// RPC calls are not allowed in Local mode.
IF stat.bLocal THEN
	RPC_MoveRel	:= M_SetRpcStatus(E_SA_RPC_ERROR.LOCAL);
	RETURN;
// Move Relative command is accepted only in OP state.
ELSIF	stat.nState <> E_SA_POS_ELT_STATE.OP	THEN
	RPC_MoveRel	:= M_SetRpcStatus(E_SA_RPC_ERROR.NOT_OP);
	RETURN;
// The positioner has to be initialised / OP (operational), i.e. already REFerenced.
ELSIF	NOT stat.bInitialised	THEN
	RPC_MoveRel	:= M_SetRpcStatus(E_SA_RPC_ERROR.CH_NOT_OP);
	RETURN;
// Set velocity cannot be 0.0.
ELSIF	in_lrVel = 0.0	THEN
	RPC_MoveRel	:= M_SetRpcStatus(E_SA_RPC_ERROR.VEL_ZERO);
	RETURN;
// Set velocity cannot be < 0.0.
ELSIF	in_lrVel <= 0.0	THEN
	RPC_MoveRel	:= M_SetRpcStatus(E_SA_RPC_ERROR.VEL_NEG);
	RETURN;
// Set velocity cannot be greater than MAX Velocity.
ELSIF	in_lrVel > cfg.lrMaxVelocity	THEN
	RPC_MoveRel	:= M_SetRpcStatus(E_SA_RPC_ERROR.VEL_MAX);
	RETURN;
// If SW limits are active, check the limits
ELSIF cfg.lrRangeLimitMax > cfg.lrRangeLimitMin THEN
	IF lrPos < cfg.lrRangeLimitMin THEN
		RPC_MoveRel	:= M_SetRpcStatus(E_SA_RPC_ERROR.SW_LIMIT_LOWER);
		RETURN;
	ELSIF lrPos > cfg.lrRangeLimitMax THEN
		RPC_MoveRel	:= M_SetRpcStatus(E_SA_RPC_ERROR.SW_LIMIT_UPPER);
		RETURN;
	END_IF
END_IF

// Set command
ctrl.nCmd	:= E_SA_CH_CMD.MOV;
ctrl.lrPos	:= lrPos;
ctrl.lrVel	:= in_lrVel;


// Call was successful
RPC_MoveRel	:= M_SetRpcStatus(E_SA_RPC_ERROR.OK);
END_METHOD

{attribute 'TcRpcEnable':='1'}
METHOD RPC_Reset : INT
VAR_INPUT
END_VAR
// If the SmarAct MCS2 Controller is in error,
// the positioner cannot be controlled.
IF stat.nCtrlErrorCode <> 0  OR  stat.nCtrlState <> E_RS_BASE_STATE.OP THEN
	RPC_Reset	:= M_SetRpcStatus(E_SA_RPC_ERROR.CTRL_ERROR);
	RETURN;
END_IF


// RPC calls are not allowed in Local mode.
IF stat.bLocal THEN
	RPC_Reset	:= M_SetRpcStatus(E_SA_RPC_ERROR.LOCAL);
	RETURN;
END_IF

// Cannot RESET positioner while moving.
IF stat.nState = E_SA_POS_ELT_STATE.OP  AND  stat.nSubstate = E_SA_POS_ELT_SUBSTATE.OP_MOVING  THEN
	RPC_Reset	:= M_SetRpcStatus(E_SA_RPC_ERROR.MOVING);
	RETURN;
END_IF


// Set command
ctrl.nCmd	:= E_SA_CH_CMD.RESET;

//stat.nState			:= E_SA_POS_ELT_STATE.NONE;
//stat.nSubstate		:= E_SA_POS_ELT_SUBSTATE.NONE;


// Call was successful
RPC_Reset	:= M_SetRpcStatus(E_SA_RPC_ERROR.OK);
END_METHOD

{attribute 'TcRpcEnable':='1'}
METHOD RPC_Stop : INT
VAR_INPUT
END_VAR
// If the SmarAct MCS2 Controller is in error,
// the positioner cannot be controlled.
IF stat.nCtrlErrorCode <> 0  OR  stat.nCtrlState <> E_RS_BASE_STATE.OP THEN
	RPC_Stop	:= M_SetRpcStatus(E_SA_RPC_ERROR.CTRL_ERROR);
	RETURN;
END_IF


// RPC calls are not allowed in Local mode.
IF stat.bLocal THEN
	RPC_Stop	:= M_SetRpcStatus(E_SA_RPC_ERROR.LOCAL);
	RETURN;
END_IF


// Set STOP command
ctrl.nCmd	:= E_SA_CH_CMD.STOP;

// Call was successful
RPC_Stop	:= M_SetRpcStatus(E_SA_RPC_ERROR.OK);
END_METHOD

END_FUNCTION_BLOCK

// ---- POUs/F_GetRpcErrorText.TcPOU
FUNCTION F_GetRpcErrorText : STRING
VAR_INPUT
	ErrorCode:	INT;
END_VAR
VAR
	str:	STRING;
END_VAR

CASE ErrorCode OF
	E_SA_RPC_ERROR.OK:					str	:= 'OK';
	E_SA_RPC_ERROR.NOT_OP:				str	:= 'Positioner not OPERATIONAL';
	E_SA_RPC_ERROR.NOT_NOTOP_READY:		str	:= 'Call failed. Not in NOTOP_READY.';
	E_SA_RPC_ERROR.NOT_NOTOP_NOTREADY:	str	:= 'Call failed. Not in NOTOP_NOTREADY/ERROR.';
	E_SA_RPC_ERROR.LOCAL:				str	:= 'RPC calls not allowed in Local mode.';
	E_SA_RPC_ERROR.SW_LIMIT_LOWER:		str	:= 'Target position beyond Lower SW Limit';
	E_SA_RPC_ERROR.SW_LIMIT_UPPER:		str	:= 'Target position beyond Upper SW Limit';
	E_SA_RPC_ERROR.CHANNEL:				str	:= 'Channel not in range [0..17]';
	E_SA_RPC_ERROR.VEL_MAX:				str	:= 'Target Velocity higher than Maximum';
	E_SA_RPC_ERROR.VEL_NEG:				str	:= 'Target Velocity cannot be negative';
	E_SA_RPC_ERROR.VEL_ZERO:			str	:= 'Target Velocity cannot be zero';
	E_SA_RPC_ERROR.CH_NOT_OP:			str	:= 'Channel not OPERATIONAL. REFerence first.';
	E_SA_RPC_ERROR.CTRL_ERROR:			str	:= 'SmarAct MCS2 Controller Problem';
	E_SA_RPC_ERROR.MOVING:				str	:= 'Positioner is moving. Stop first.';
	E_SA_RPC_ERROR.COMM:				str	:= 'SmarAct MCS2 Controller Communication Problem';
ELSE
	str	:= 'Unregistered RPC error.';
END_CASE

F_GetRpcErrorText	:= str;

END_FUNCTION

// ---- POUs/F_STRING_TO_LINT.TcPOU
FUNCTION F_STRING_TO_LINT : LINT
VAR_INPUT
	in_s:	STRING;
END_VAR
VAR
	lrVal:	LREAL;
END_VAR

// STRING_TO_LINT DOES NOT WORK !!!!!
//
// The string has to be converted to LREAL first and then to LINT
//
lrVal	:= STRING_TO_LREAL(in_s);

F_STRING_TO_LINT	:= LREAL_TO_LINT(lrVal);

END_FUNCTION

// ---- Examples/FB_SA_CH_PDS_IRIS.TcPOU
FUNCTION_BLOCK FB_SA_CH_PDS_IRIS EXTENDS FB_SA_CHANNEL_BASE
VAR_INPUT
END_VAR
VAR_OUTPUT
END_VAR
VAR
END_VAR

//
// SID-50 specific non-linear conversion 
// from Device units [nd] to user units [%] of opening.
//
METHOD M_ConvertPosDev2User : LREAL
VAR_INPUT
	lnDevValue:	LINT;
END_VAR
VAR
	lrDiam:	LREAL;		// Diameter of opening [mm].
END_VAR
//
// Note that iris increases the opening when moving in negative direction.
// That's why the scale is negative in the configuration.
// Linear conversion implemented in M_ConvertDev2User().
// UU   = DevU / scale * BASE_RES
// DevU = UU   * scale / BASE_RES
//
lrDiam	:= M_ConvertDev2User(lnDevValue);

//
// Maximum opening is 50 mm.
// Current opening is relative to that.
//    % = diam^2 / 50^2 * 100.0
//
M_ConvertPosDev2User := (lrDiam * lrDiam) / (50.0 * 50.0) * 100.0;
END_METHOD

//
// SID-50 specific non-linear conversion 
// from user units [%] of opening to Device units [nd].
//
METHOD M_ConvertPosUser2Dev : LINT
VAR_INPUT
	lrUserValue:	LREAL;	// Percentage of opening
END_VAR
VAR
	lrDiam:	LREAL;		// Diameter of opening [mm].
END_VAR
//
// Note that iris increases the opening when moveng in negative direction.
// That's why the scale is negative in the configuration.
//

//
// Get the opening diameter from the percentage relative to 50 mm for SID-50.
//    % = lrUserValue;
//    % = 100.0 * diam^2 / 50^2  ==> diam = SQRT(% / 100.0 * 50^2)
//
lrDiam	:= SQRT(lrUserValue / 100.0 * 50.0 * 50.0);

//
// Convert diameter to device unitd - linear conversion.
//
M_ConvertPosUser2Dev := M_ConvertUser2Dev(lrDiam);
END_METHOD

END_FUNCTION_BLOCK

// ---- Examples/FB_SMARACT_SIM.TcPOU
FUNCTION_BLOCK FB_SMARACT_SIM EXTENDS FB_SMAR_ACT_BASE
VAR_INPUT
END_VAR
VAR_OUTPUT
END_VAR
VAR
	//
	// TODO USER: Add existing SmarAct Positioners
	//
	// We use prefix 'x_' just for the convenience that
	// all positioners appear together in the OPC UA Namespace.
	//
	x_fw1:	FB_SA_CHANNEL_BASE;	// CH 0
	x_fw2:	FB_SA_CHANNEL_BASE;	// CH 1
	x_iris:	FB_SA_CH_PDS_IRIS;	// CH 2 non-linear scaling for % of opening
END_VAR

//
// Execute the base class object FB_SMAR_ACT_BASE.
//
SUPER^();

METHOD M_ConfigureUser
VAR_INPUT
END_VAR
VAR
	i:		UINT;
	nMod:	UINT;	// Module number
	
END_VAR
//
// This method defines specific configurations for each positioner/channel.
//

// 
// In this example, three positioners are defined in FB_SMARACT_SIM.
//
//	fw1:	FB_SA_CHANNEL_BASE;
//	fw2:	FB_SA_CHANNEL_BASE;
//	iris:	FB_SA_CHANNEL_BASE;
//

//
// Configure used channels [0..17].
// In this example, there are three used channels: 0, 1 and 2.
//
cfg.arrUsedCh[0]	:= TRUE;
cfg.arrUsedCh[1]	:= TRUE;
cfg.arrUsedCh[2]	:= TRUE;


//
// Set pointers to instances of used channels
//
ptrCH[0]	:= ADR(x_fw1);
ptrCH[1]	:= ADR(x_fw2);
ptrCH[2]	:= ADR(x_iris);


//
// Initial configuration of each exiting positioner.
//

//
// SFW-6-25.4 - Filter Wheel 1
//
x_fw1.M_Configure(
	in_sName			:= 'Filter Wheel - 1',
	in_sUnits			:= 'deg',
	in_lrScale			:= 1.0, 
	in_lrREF_POS		:= 60.0,	// REF mark pos
	in_lrREF_VEL		:= 20.0,	// Velocity for referencing [UU/s]
	in_nHOLD			:= -1,		// Hold infinitely
	in_lrINP_THR		:= 0.001,	// in-pos threshold = 0.001 deg
	in_nINP_DEL			:= 500,		// in-pos delay 500 ms
	in_lrMaxVelocity	:= 30,		// Maximum permitted Velocity
	in_lrRangeLimitMin	:= 0.0,		// Min=Max ==> No limits
	in_lrRangeLimitMax	:= 0.0,		// Min=Max ==> No limits 
	in_nREF_OPT			:= 0,		// Referencing in positive direction
	in_nCAL_OPT			:= 0,		// Calibrating in positive direction
	in_nPCON_OPT		:= 256);	// 'in-pos' flag set

//
// SFW-6-25.4 - Filter Wheel 2
//
x_fw2.M_Configure(
	in_sName			:= 'Filter Wheel - 2',
	in_sUnits			:= 'deg',
	in_lrScale			:= 1.0, 
	in_lrREF_POS		:= 120.0,	// REF mark pos
	in_lrREF_VEL		:= 20.0,	// Velocity for referencing [UU/s]
	in_nHOLD			:= -1,		// Hold infinitely
	in_lrINP_THR		:= 0.001,	// in-pos threshold = 0.001 deg
	in_nINP_DEL			:= 1000,	// in-pos delay 500 ms
	in_lrMaxVelocity	:= 30,		// Maximum permitted Velocity
	in_lrRangeLimitMin	:= 0.0,		// Min=Max ==> No limits
	in_lrRangeLimitMax	:= 0.0,		// Min=Max ==> No limits 
	in_nREF_OPT			:= 0,		// Referencing in positive direction
	in_nCAL_OPT			:= 0,		// Calibrating in positive direction
	in_nPCON_OPT		:= 256);	// 'in-pos' flag set

//
// SID-50 - Iris Diaphragm
//
// Note: Because the scale is negative, MIN and MAX values are swapped.
//       In Device Units, the diaphragm will move between -5..-50 (/scale) mm.
//       In User   Units, the diaphragm will move between 1..100 %.
//
// The position of the diaphragm is the percentage of the opening.
//

x_iris.M_Configure(
	in_sName			:= 'SHAPS Diaphragm',
	in_sUnits			:= '%',
	in_lrScale			:= -0.001763245, 
	in_lrREF_POS		:= 34.33,	// REF mark pos in %. (Diam = 29.29832067 mm)
	in_lrREF_VEL		:= 5.0,		// Velocity for referencing [UU/s]
	in_nHOLD			:= -1,		// Hold infinitely
	in_lrINP_THR		:= 0.0005,	// in-pos threshold = 0.0005 %
	in_nINP_DEL			:= 500,		// in-pos delay 500 ms
	in_lrMaxVelocity	:= 15,		// Maximum permitted Velocity
	in_lrRangeLimitMin	:= 100.001,	// Min limit (positive because in_lrScale < 0) !!!
	in_lrRangeLimitMax	:= 0.999,	// Max limit (negative because in_lrScale < 0) !!!
	in_nREF_OPT			:= 0,		// Referencing in positive direction
	in_nCAL_OPT			:= 0,		// Calibrating in positive direction
	in_nPCON_OPT		:= 256);	// 'in-pos' flag set
END_METHOD

END_FUNCTION_BLOCK

// ---- POUs/Simulation/FB_SIM_SMAR_ACT.TcPOU
FUNCTION_BLOCK FB_SIM_SMAR_ACT EXTENDS FB_SIM_TCP_DEVICE_BASE
VAR_INPUT
END_VAR
VAR_OUTPUT
END_VAR
VAR
	arrCH:		ARRAY [0..17] OF FB_SIM_SA_CHANNEL;
	i:			UINT;
END_VAR

IF NOT in_bEnable THEN
	RETURN;
ELSE
	//
	// Execute instance of the simulator
	//
	Device(	in_bSimulation	:= in_bSimulation,
			in_sTcpIpAdr	:= in_sTcpIpAdr,
			in_nTcpPort		:= in_nTcpPort);
	
	//
	// Execute State Machine for each instance Channel simulator.
	//
	FOR i:=0 TO 17 DO
		arrCH[i].M_StateMachine();
	END_FOR
			
	//
	// Check for received commands.
	//
	IF Device.out_bAccepted AND Device.out_bReceived THEN
		// A command has arrived. Send a simulated reply
		sReply	:=	M_GetSimReply(in_sReceived	:=Device.out_sReceived); 
		
		// Trigger SEND only if there is a reply
		IF sReply <> ''	THEN
			ptrDevCtrl^.nCommand	:= E_RS_COMM_CMD.SEND;
			ptrDevCtrl^.sCmd		:= sReply;
			ptrDevCtrl^.bExecute	:= TRUE;
		END_IF
	END_IF
END_IF

METHOD M_GetSimReply : STRING(255)
VAR_INPUT
	{attribute 'OPC.UA.DA' := '0'}
	in_sReceived:	STRING(255);		// String received from a client
END_VAR
VAR
	sReply:	STRING(255);
	sTmp:	STRING;
	sTmp2:	STRING;
	lrVal:	LREAL;
	nValue:	UINT;
	i:		INT;
    fbFormat   : FB_FormatString;
    sOut       : T_MaxString;
	nCh:	UINT;	// Channel number
	nPos:	INT;	// Position in the string

	lnVel:	LINT;	// MOVE Velocity
	lnPos:	LINT;	// MOVE Target Position
END_VAR
//
// Commands related to the controller/DEVice
//
IF FIND (in_sReceived, '*IDN?') > 0 THEN
	// MCS2 ID
	M_GetSimReply	:= CONCAT('SIM SmarAct;MCS2-00005855;MCS2-00005855;07/05/21', in_sReplySuffix);

ELSIF FIND (in_sReceived, ':DEV:SNUM?') > 0 THEN
	// MCS2 S/N
	M_GetSimReply	:= CONCAT('"MCS2-00005855"', in_sReplySuffix);

ELSIF FIND (in_sReceived, ':DEV:STAT?') > 0 THEN
	// MCS2 State
	// 16 => Only stDevState.bGLOBAL_INPUT set to TRUE.
	M_GetSimReply	:= CONCAT('16', in_sReplySuffix);

//
// Replies to commands starting with ':MOD'.
//
ELSIF FIND(in_sReceived, ':MOD') = 1 THEN
	IF FIND(in_sReceived, ':STAT?') > 1 THEN
		// MOD state is 1 - BIT_SM_PRESENT.
		M_GetSimReply	:= CONCAT('1', in_sReplySuffix);
	END_IF

ELSE
	//
	// Commands related to individual channels
	//
	IF	FIND (in_sReceived, ':CHAN') = 1	THEN
			// Get the channel number that comes 
			// after ':CHAN', e.g. ':CHAN2:STAT?'
			sTmp	:= DELETE(in_sReceived,5,1);
			nCh		:= STRING_TO_UINT(sTmp);
			// The string looks like '2:STAT?' now.
			// Remove the channel number and the following ':' from the command,
			// i.e. remove '2:' and pass 'STAT?' to the channel.
			nPos	:= FIND (sTmp, ':');
			sTmp	:= DELETE(sTmp,nPos,1);
			sReply	:= arrCH[nCH].M_GetChSimReply(sTmp);
			IF sReply <> ''	THEN
				// There is a reply from the channel.
				// Channel reply doesn't contain the reply suffix. Add it.
				M_GetSimReply	:= CONCAT(sReply, in_sReplySuffix);
			ELSE
				// Channel Reply is empty string.
				// Don't reply, i.e. reply is empty string.
				M_GetSimReply	:= '';
			END_IF
	ELSIF	FIND (in_sReceived, ':REF') = 1	THEN
			// Get the channel number that comes 
			// after ':REF' , e.g. ':REF2'
			sTmp	:= DELETE(in_sReceived,4,1);
			nCh		:= STRING_TO_UINT(sTmp);
			arrCH[nCH].M_StartREF();
			M_GetSimReply	:= '';	// No reply to this command
	ELSIF	FIND (in_sReceived, ':CAL') = 1		THEN
			// Get the channel number that comes 
			// after ':CAL', e.g. ':CAL2'
			sTmp	:= DELETE(in_sReceived,4,1);
			nCh		:= STRING_TO_UINT(sTmp);
			arrCH[nCH].M_StartCAL();
			M_GetSimReply	:= '';	// No reply to this command
	ELSIF	FIND (in_sReceived, ':MOVE') = 1	THEN
			// Get the channel number that comes 
			// after ':MOVE', in e.g. ':MOVE2 100000'
			sTmp	:= DELETE(in_sReceived,5,1);	// '2 100000'
			nCh		:= STRING_TO_UINT(sTmp);
			// Find the space and delete everything up to and including the space.
			nPos	:= FIND (sTmp, ' ');
			sTmp2	:= DELETE(sTmp, nPos, 1);	// '100000'
			lnPos	:= F_STRING_TO_LINT(sTmp2);	// Target Position
			lnVel	:= arrCH[nCH].ctrl.lnVEL;	// Target Velocity
			arrCH[nCH].M_StartMOVE(lnPos, lnVel);
			M_GetSimReply	:= '';	// No reply to this command
	ELSIF	FIND (in_sReceived, ':STOP') = 1	THEN
			// Get the channel number that comes 
			// after ':MOVE', e.g. ':MOVE2'
			sTmp	:= DELETE(in_sReceived,5,1);
			nCh		:= STRING_TO_UINT(sTmp);
			arrCH[nCH].M_STOP();
			M_GetSimReply	:= '';	// No reply to this command
	END_IF
END_IF
END_METHOD

END_FUNCTION_BLOCK

// ---- POUs/Simulation/FB_SIM_SA_CHANNEL.TcPOU
FUNCTION_BLOCK FB_SIM_SA_CHANNEL
VAR_INPUT
END_VAR
VAR_OUTPUT
END_VAR
VAR
	cfg:	T_SA_SIM_CH_CFG;
	ctrl:	T_SA_SIM_CH_CTRL;
	stat:	T_SA_SIM_CH_STATUS;
	
	fbTimer:		TON;

END_VAR

// Execute State Machine
M_StateMachine();

METHOD M_GetChSimReply : STRING(255)
VAR_INPUT
	{attribute 'OPC.UA.DA' := '0'}
	in_sCmd:	STRING(255);		// String received from a client
END_VAR
VAR
	sReply:	STRING(255);
	sTmp:	STRING;
	lrVal:	LREAL;
	nValue:	UINT;
	i:		INT;
    fbFormat   : FB_FormatString;
    sOut       : T_MaxString;
	nCh:	INT := 8;	// Number of channels for models 218 and 224
END_VAR

IF FIND (in_sCmd, '?') > 0 THEN
	// This is a query command.
	// There is a reply.
	// Check commands one by one.

	IF FIND (in_sCmd, 'STAT?') > 0 THEN
		// Channel state
		M_GetChSimReply	:= UDINT_TO_STRING(stat.nSTATE);
	ELSIF FIND (in_sCmd, 'CAL:OPT?') > 0 THEN
		// Channel state
		M_GetChSimReply	:= UINT_TO_STRING(cfg.nCAL_OPT);
	ELSIF FIND (in_sCmd, 'REF:OPT?') > 0 THEN
		// Channel state
		M_GetChSimReply	:= UINT_TO_STRING(cfg.nREF_OPT);
	ELSIF FIND (in_sCmd, 'PCON:OPT?') > 0 THEN
		// Channel Positioner control otions
		M_GetChSimReply	:= UINT_TO_STRING(cfg.nPCON_OPT);
	ELSIF FIND (in_sCmd, 'INP:THR?') > 0 THEN
		// Channel in-position threshold
		M_GetChSimReply	:= UDINT_TO_STRING(cfg.nINP_THR);
	ELSIF FIND (in_sCmd, 'INP:DEL?') > 0 THEN
		// Channel in-position delay
		M_GetChSimReply	:= UDINT_TO_STRING(cfg.nINP_DEL);
	ELSIF FIND (in_sCmd, 'RLIM:MIN?') > 0 THEN
		// Channel Limit Min
		M_GetChSimReply	:= LINT_TO_STRING(cfg.lnRLIM_MIN);
	ELSIF FIND (in_sCmd, 'RLIM:MAX?') > 0 THEN
		// Channel Limit Max
		M_GetChSimReply	:= LINT_TO_STRING(cfg.lnRLIM_MAX);
	ELSIF FIND (in_sCmd, 'POS:TARG?') > 0 THEN
		// Channel target position
		M_GetChSimReply	:= LINT_TO_STRING(stat.lnPosTarget);
	ELSIF FIND (in_sCmd, 'POS:CURR?') > 0 THEN
		// Channel actual position
		M_GetChSimReply	:= LINT_TO_STRING(stat.lnPosActual);
	ELSIF FIND (in_sCmd, 'CLIN?') > 0 THEN
		// Channel 
		M_GetChSimReply	:= DINT_TO_STRING(cfg.nCLIN);
	ELSIF FIND (in_sCmd, 'TUN:BASE:UNIT?') > 0 THEN
		// Channel 
		M_GetChSimReply	:= DINT_TO_STRING(cfg.nBASE_UNIT);
	ELSIF FIND (in_sCmd, 'TUN:BASE:RES?') > 0 THEN
		// Channel 
		M_GetChSimReply	:= DINT_TO_STRING(cfg.nBASE_RES);
	ELSIF FIND (in_sCmd, 'TUN:MTYP?') > 0 THEN
		// Channel 
		M_GetChSimReply	:= DINT_TO_STRING(cfg.nTUN_MTYP);
	ELSIF FIND (in_sCmd, 'TUN:RTYP?') > 0 THEN
		// Channel 
		M_GetChSimReply	:= LINT_TO_STRING(cfg.nTUN_RTYP);
	END_IF
ELSE
	// This is a control command.
	// There is NO reply.
	// BUT there are some action to be taken

	IF FIND (in_sCmd, 'CAL:OPT ') > 0 THEN
		// Get the value
		sTmp			:= DELETE(in_sCmd,8,1);
		cfg.nCAL_OPT	:= STRING_TO_UINT(sTmp);
	ELSIF FIND (in_sCmd, 'REF:OPT ') > 0 THEN
		// Get the value
		sTmp			:= DELETE(in_sCmd,8,1);
		cfg.nREF_OPT	:= STRING_TO_UINT(sTmp);
	ELSIF FIND (in_sCmd, 'PCON:OPT ') > 0 THEN
		// Get the value
		sTmp			:= DELETE(in_sCmd,9,1);
		cfg.nPCON_OPT	:= STRING_TO_UINT(sTmp);
	ELSIF FIND (in_sCmd, 'INP:THR ') > 0 THEN
		// Get the value
		sTmp			:= DELETE(in_sCmd,8,1);
		cfg.nINP_THR	:= STRING_TO_UDINT(sTmp);
	ELSIF FIND (in_sCmd, 'INP:DEL ') > 0 THEN
		// Get the value
		sTmp			:= DELETE(in_sCmd,8,1);
		cfg.nINP_DEL	:= STRING_TO_UDINT(sTmp);
	ELSIF FIND (in_sCmd, 'RLIM:MIN ') > 0 THEN
		// Get the value
		sTmp			:= DELETE(in_sCmd,9,1);
		cfg.lnRLIM_MIN	:= STRING_TO_UINT(sTmp);
	ELSIF FIND (in_sCmd, 'RLIM:MAX ') > 0 THEN
		// Get the value
		sTmp			:= DELETE(in_sCmd,9,1);
		cfg.lnRLIM_MAX	:= STRING_TO_UINT(sTmp);
	ELSIF FIND (in_sCmd, 'POS:TARG ') > 0 THEN
		// Get the value
		sTmp			:= DELETE(in_sCmd,9,1);
		stat.lnPosTarget:= F_STRING_TO_LINT(sTmp);
	ELSIF FIND (in_sCmd, 'POS:CURR ') > 0 THEN
		// Get the value
		sTmp			:= DELETE(in_sCmd,9,1);
		stat.lnPosActual:= F_STRING_TO_LINT(sTmp);
	ELSIF FIND (in_sCmd, 'VEL ') > 0 THEN
		// Get the value
		sTmp			:= DELETE(in_sCmd,4,1);
		cfg.lnVEL		:= F_STRING_TO_LINT(sTmp);
		ctrl.lnVEL		:= F_STRING_TO_LINT(sTmp);
	ELSIF FIND (in_sCmd, 'POS ') > 0 THEN
		// Get the value
		sTmp			:= DELETE(in_sCmd,4,1);
		stat.lnPosActual:= F_STRING_TO_LINT(sTmp);
	END_IF
	
	// There is no reply to control commands !!!
	M_GetChSimReply	:= '';
END_IF
END_METHOD

METHOD M_StartCAL
VAR_INPUT
END_VAR
// Start CALibration simulation
;
END_METHOD

METHOD M_StartMOVE
VAR_INPUT
	in_lnPos:	LINT;	// Target Position
	in_lnVel:	LINT;	// Target Velocity
END_VAR
VAR 
	nState:		UDINT := 0;
	nTime:		UDINT :=0;	// Calculated move time [ms].
END_VAR
// Start MOVE simulation

// Set target velocity and position.
ctrl.lnVEL			:= in_lnVel;
ctrl.lnPOS			:= in_lnPos;
stat.lnPosTarget	:= in_lnPos;
stat.lnPosStart		:= stat.lnPosActual;	// MOVE started from this position

// Get the distance to move.
// If distance is zero, do nothing.
stat.lnDistance	:= ctrl.lnPOS - stat.lnPosActual;
IF stat.lnDistance = 0	THEN
	// No movement
	fbTimer(IN:=FALSE);
	RETURN;
END_IF

nState	:= nState OR E_SA_CH_STATE.BIT_ACTIVELY_MOVING;
nState	:= nState OR E_SA_CH_STATE.BIT_CLOSED_LOOP_ACTIVE;
nState	:= nState OR E_SA_CH_STATE.BIT_SENSOR_PRESENT;
nState	:= nState OR E_SA_CH_STATE.BIT_IS_CALIBRATED;
nState	:= nState OR E_SA_CH_STATE.BIT_IS_REFERENCED;
nState	:= nState OR E_SA_CH_STATE.BIT_AMPLIFIER_ENABLED;

stat.nSTATE	:= nState;

// Get time [ms] needed for the move
IF in_lnVel = 0	THEN
	nTime	:= 1000;
ELSE	
	nTime	:= LINT_TO_UDINT(1000 * ABS(stat.lnDistance) / in_lnVel);
END_IF

IF nTime > 0 THEN
	// Set the positioner State Machine State
	stat.nPosState	:=	E_SA_POS_SM_STATE.MOVING;
	
	// Start the timer.
	// Simulated REFerencing should finish in 5 sec.
	fbTimer(IN:=FALSE);
	fbTimer(IN:=TRUE,PT:=UDINT_TO_TIME(nTime));
ELSE
	// No movement
	fbTimer(IN:=FALSE);
END_IF
END_METHOD

METHOD M_StartREF
VAR_INPUT
END_VAR
VAR 
	nState:		UDINT := 0;
END_VAR
// Start REFerencing simulation

nState	:= nState OR E_SA_CH_STATE.BIT_ACTIVELY_MOVING;
nState	:= nState OR E_SA_CH_STATE.BIT_CLOSED_LOOP_ACTIVE;
nState	:= nState OR E_SA_CH_STATE.BIT_REFERENCING;
nState	:= nState OR E_SA_CH_STATE.BIT_SENSOR_PRESENT;
nState	:= nState OR E_SA_CH_STATE.BIT_AMPLIFIER_ENABLED;

stat.nSTATE	:= nState;

// Set the positioner State Machine State
stat.nPosState	:=	E_SA_POS_SM_STATE.CALIB_REF;

// Start the timer.
// Simulated REFerencing should finish in 5 sec.
fbTimer(IN:=FALSE);
fbTimer(IN:=TRUE,PT:=T#5S);
END_METHOD

METHOD M_StateMachine
VAR_INPUT
END_VAR
VAR 
	nState:		UDINT := 0;
	lrProgress:	LREAL;		// Movement progress [0.0..1.0]
	lnPosInc:	LINT;		// Position increment from starting position.
END_VAR
// Execute the timer.
fbTimer();

CASE stat.nPosState OF
	E_SA_POS_SM_STATE.CALIB_REF:
		// Check if referencing is complete.
		IF fbTimer.Q THEN
			// Reset timer
			fbTimer(IN:=FALSE);
			// Set flags for completed REFerencing
			nState	:= nState OR E_SA_CH_STATE.BIT_CLOSED_LOOP_ACTIVE;
			nState	:= nState OR E_SA_CH_STATE.BIT_SENSOR_PRESENT;
			nState	:= nState OR E_SA_CH_STATE.BIT_IS_CALIBRATED;
			nState	:= nState OR E_SA_CH_STATE.BIT_IS_REFERENCED;
			nState	:= nState OR E_SA_CH_STATE.BIT_REFERENCE_MARK;
			nState	:= nState OR E_SA_CH_STATE.BIT_AMPLIFIER_ENABLED;
			nState	:= nState OR E_SA_CH_STATE.BIT_IN_POSITION;
			
			stat.nSTATE	:= nState;
			
			// Set the calibrated position
			stat.lnPosTarget	:= cfg.lnREF_POS;
			stat.lnPosActual	:= cfg.lnREF_POS;
			
			// Set the positioner State Machine State
			stat.nPosState	:=	E_SA_POS_SM_STATE.OP;
		END_IF
	E_SA_POS_SM_STATE.MOVING:
		// Simulate movement progress
		IF fbTimer.PT = T#0MS THEN
			RETURN;
		END_IF
		lrProgress	:= TIME_TO_LREAL(fbTimer.ET) / TIME_TO_LREAL(fbTimer.PT);
		lnPosInc	:= LREAL_TO_LINT(LINT_TO_LREAL(stat.lnDistance) * lrProgress);
		stat.lnPosActual	:= stat.lnPosStart + lnPosInc;
		
		// Check if the move is complete.
		IF fbTimer.Q THEN
			// Reset timer
			fbTimer(IN:=FALSE);
			// Set flags for completed REFerencing
			nState	:= nState OR E_SA_CH_STATE.BIT_CLOSED_LOOP_ACTIVE;
			nState	:= nState OR E_SA_CH_STATE.BIT_SENSOR_PRESENT;
			nState	:= nState OR E_SA_CH_STATE.BIT_IS_CALIBRATED;
			nState	:= nState OR E_SA_CH_STATE.BIT_IS_REFERENCED;
			nState	:= nState OR E_SA_CH_STATE.BIT_AMPLIFIER_ENABLED;
			nState	:= nState OR E_SA_CH_STATE.BIT_IN_POSITION;
			
			stat.nSTATE	:= nState;
			
			// Set the positioner State Machine State
			stat.nPosState	:=	E_SA_POS_SM_STATE.OP;
		END_IF
END_CASE
END_METHOD

METHOD M_STOP
VAR_INPUT
END_VAR
VAR 
	nState:		UDINT := 0;
END_VAR
// STOP MOVE simulation
// Start MOVE simulation

// No movement. Stop the timer.
fbTimer(IN:=FALSE);

nState	:= nState OR E_SA_CH_STATE.BIT_CLOSED_LOOP_ACTIVE;
nState	:= nState OR E_SA_CH_STATE.BIT_SENSOR_PRESENT;
nState	:= nState OR E_SA_CH_STATE.BIT_IS_CALIBRATED;
nState	:= nState OR E_SA_CH_STATE.BIT_IS_REFERENCED;
nState	:= nState or E_SA_CH_STATE.BIT_AMPLIFIER_ENABLED;

stat.nSTATE	:= nState;

stat.nPosState	:=	E_SA_POS_SM_STATE.OP;
END_METHOD

END_FUNCTION_BLOCK

// ---- GlobalTextList.TcGTLO
TEXTLIST GlobalTextList
  504 = '%.1f'
  771 = '%.2f'
  615 = '%.3f'
  361 = '%.3f W'
  955 = '%s'
  280 = 'Actual Position [UU]'
  817 = 'Amplifier Enabled'
  740 = 'Bolometer'
  232 = 'Bolometer Range'
  689 = 'Calibrated'
  186 = 'Calibrating'
  354 = 'CH0 Positioner'
  527 = 'CH1 Positioner'
  317 = 'CH2 Positioner'
  421 = 'Channel State'
  170 = 'Device State'
  767 = 'Device Status'
  64 = 'Device Substate'
  378 = 'DISABLE'
  608 = 'ENABLE'
  144 = 'Enabled'
  785 = 'End Stop'
  529 = 'Error'
  806 = 'Error Text'
  760 = 'Following Error'
  107 = 'GREEN if initialised'
  194 = 'If GREEN, last ZERO SAVE was successfull'
  653 = 'In Position'
  963 = 'INIT'
  973 = 'Limit Reached'
  648 = 'Local Control'
  172 = 'Loop Active'
  501 = 'Measured power [W]'
  217 = 'MOVE'
  852 = 'MOVE ABS'
  349 = 'Move Delayed'
  391 = 'MOVE REL'
  362 = 'Movement Failed'
  340 = 'Moving'
  390 = 'On Reference'
  292 = 'Overload'
  883 = 'Overtemperature'
  518 = 'Phased'
  150 = 'Pos [UU]'
  499 = 'Pos [UU]: '
  952 = 'Positioner Device State'
  786 = 'Positioner Device Substate'
  331 = 'Positioner Fault'
  283 = 'Positioner Status'
  477 = 'Positioner User Units'
  275 = 'Referenced'
  742 = 'Referencing'
  989 = 'Rel Pos [UU]: '
  787 = 'RESET'
  350 = 'RPC Status:'
  772 = 'Selected Positioner'
  755 = 'Sensor Present'
  610 = 'Set Position Offset [UU]'
  784 = 'Set Position [UU]'
  924 = 'Set Velocity [UU/s]'
  839 = 'SmarAct Library Version'
  277 = 'Start Zeroing process'
  701 = 'State'
  233 = 'State:'
  298 = 'Status'
  82 = 'Status:'
  493 = 'STOP'
  553 = 'Streaming'
  450 = 'Substate'
  492 = 'Substate:'
  171 = 'Vel [UU/s'
  140 = 'Vel [UU/s]'
  219 = 'Vel [UU/s]: '
  930 = 'Ver. %s'
  813 = 'ZERO'
END_TEXTLIST

// ---- VISUs/GUIs/GUI_SmarAct_PDS.TcVIS
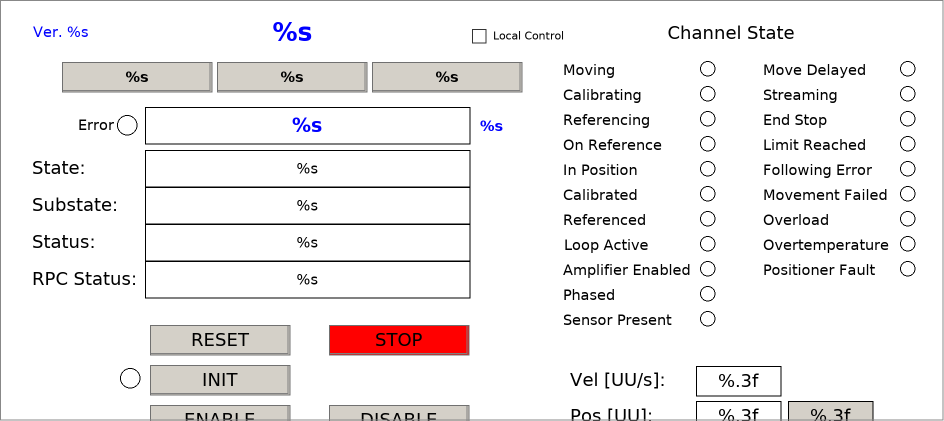
VISUALIZATION GUI_SmarAct_PDS  // 944x421
    Frame (0,0 944x421)
        shows GUI_TEMPLATE_SMAR_ACT(m_Instance := MAIN.SmarAct_PDS)
END_VISUALIZATION

// ---- VISUs/GUIs/GUI_SmarAct_SIM.TcVIS
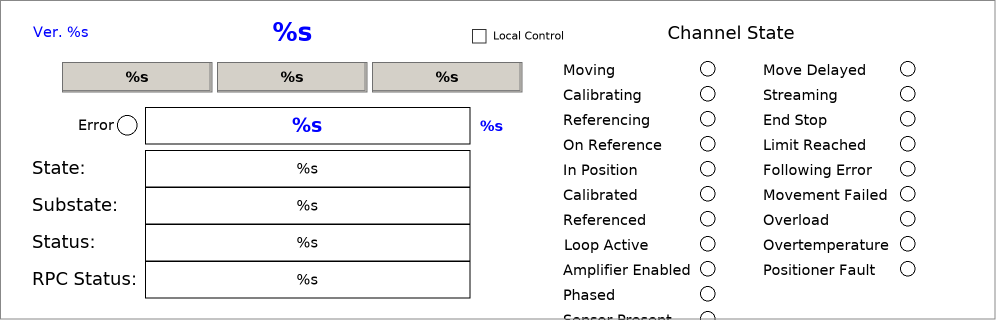
VISUALIZATION GUI_SmarAct_SIM  // 996x320
    Frame (0,0 996x320)
        shows GUI_TEMPLATE_SMAR_ACT(m_Instance := MAIN.SmarAct_Sim)
END_VISUALIZATION

// ---- VISUs/Templates/GUI_TEMPLATE_SMAR_ACT.TcVIS
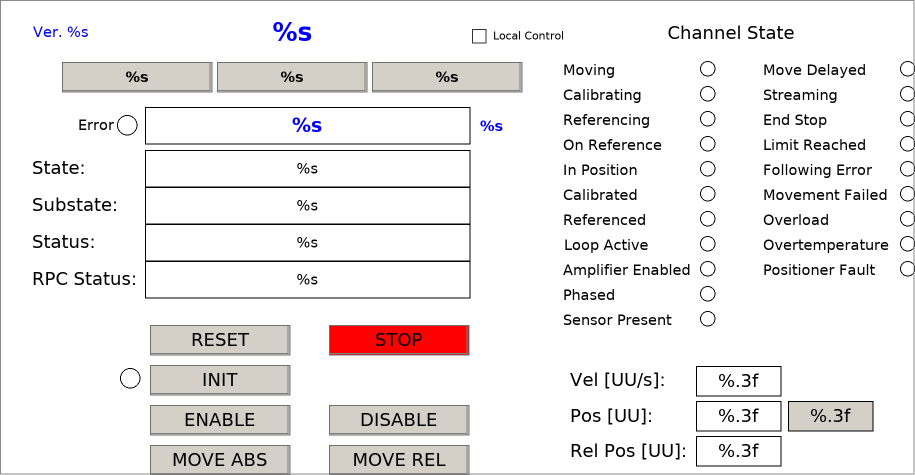
VISUALIZATION GUI_TEMPLATE_SMAR_ACT  // 915x475
VAR_IN_OUT
	m_Instance:	FB_SMAR_ACT_BASE;
END_VAR
    Rectangle (145,107 325x37), "%s", tooltip "Selected Positioner", text variable: m_Instance.ptrGuiCH^.cfg.sName
    Button (62,62 150x30), "%s", tooltip "CH0 Positioner", text variable: m_Instance.arrChName[0]
        OnMouseClick: execute { m_Instance.nGuiIndex := 0; }
    Button (217,62 150x30), "%s", tooltip "CH1 Positioner", text variable: m_Instance.arrChName[1], input disabled if: m_Instance.ptrCH[1] = 0
        OnMouseClick: execute { m_Instance.nGuiIndex := 1; }
    Button (372,62 150x30), "%s", tooltip "CH2 Positioner", text variable: m_Instance.arrChName[2], input disabled if: m_Instance.ptrCH[2] = 0
        OnMouseClick: execute { m_Instance.nGuiIndex := 2; }
    Button (150,365 140x30), "INIT", input disabled if: NOT m_Instance.ptrGuiCH^.stat.bLocal OR m_Instance.ptrGuiCH^.stat.bInitialised
        OnMouseClick: execute { m_Instance.ptrGuiCH^.ctrl.nCmd:=E_SA_CH_CMD.REF; }
    Button (150,445 140x30), "MOVE ABS", input disabled if: NOT m_Instance.ptrGuiCH^.stat.bLocal OR m_Instance.ptrGuiCH^.stat.nState <> E_SA_POS_ELT_STATE.OP
        OnMouseClick: execute { m_Instance.ptrGuiCH^.ctrl.nCmd:=E_SA_CH_CMD.MOV; }
    Rectangle (696,366 85x30), "%.3f", tooltip "Set Velocity [UU/s]", text variable: m_Instance.ptrGuiCH^.ctrl.lrVel
        OnMouseClick: write the text variable via Default
    Label (567,365 100x30), "Vel [UU/s]:"
    Label (567,401 100x30), "Pos [UU]:"
    Rectangle (696,401 85x30), "%.3f", tooltip "Set Position [UU]", text variable: m_Instance.ptrGuiCH^.ctrl.lrPos
        OnMouseClick: write the text variable via Default
    Rectangle (788,401 85x30), "%.3f", tooltip "Actual Position [UU]", text variable: m_Instance.ptrGuiCH^.stat.lrPosActual
    Button (329,325 140x30), "STOP"
        OnMouseClick: execute { m_Instance.ptrGuiCH^.ctrl.nCmd:=E_SA_CH_CMD.STOP; }
    Rectangle (120,12 345x39), "%s", text variable: m_Instance.in_sName
    Label (560,55 140x30), "Moving"
    Label (561,230 140x30), "Loop Active"
    Label (560,80 140x30), "Calibrating"
    Label (560,105 140x30), "Referencing"
    Label (560,305 140x30), "Sensor Present"
    Label (560,180 140x30), "Calibrated"
    Label (560,205 140x30), "Referenced"
    Label (760,105 140x30), "End Stop"
    Label (760,130 140x30), "Limit Reached"
    Label (560,130 140x30), "On Reference"
    Label (560,255 140x30), "Amplifier Enabled"
    Label (560,155 140x30), "In Position"
    Label (75,110 43x30), "Error"
    Ellipse (700,61 15x15), colour toggle: m_Instance.ptrGuiCH^.stat.stState.bACTIVELY_MOVING
    Ellipse (700,236 15x15), colour toggle: m_Instance.ptrGuiCH^.stat.stState.bCLOSED_LOOP_ACTIVE
    Ellipse (700,86 15x15), colour toggle: m_Instance.ptrGuiCH^.stat.stState.bCALIBRATING
    Ellipse (700,111 15x15), colour toggle: m_Instance.ptrGuiCH^.stat.stState.bREFERENCING
    Ellipse (700,311 15x15), colour toggle: m_Instance.ptrGuiCH^.stat.stState.bSENSOR_PRESENT
    Ellipse (700,186 15x15), colour toggle: m_Instance.ptrGuiCH^.stat.stState.bIS_CALIBRATED
    Ellipse (700,211 15x15), colour toggle: m_Instance.ptrGuiCH^.stat.stState.bIS_REFERENCED
    Ellipse (900,111 15x15), colour toggle: m_Instance.ptrGuiCH^.stat.stState.bEND_STOP_REACHED
    Ellipse (900,136 15x15), colour toggle: m_Instance.ptrGuiCH^.stat.stState.bRANGE_LIMIT_REACHED
    Ellipse (700,136 15x15), colour toggle: m_Instance.ptrGuiCH^.stat.stState.bREFERENCE_MARK
    Ellipse (700,261 15x15), colour toggle: m_Instance.ptrGuiCH^.stat.stState.bAMPLIFIER_ENABLED
    Ellipse (700,161 15x15), colour toggle: m_Instance.ptrGuiCH^.stat.stState.bIN_POSITION
    Ellipse (117,115 20x20), colour toggle: m_Instance.ptrGuiCH^.stat.bError
    Label (760,155 140x30), "Following Error"
    Ellipse (900,161 15x15), colour toggle: m_Instance.ptrGuiCH^.stat.stState.bFOLLOWING_LIMIT_REACHED
    Label (760,180 140x30), "Movement Failed"
    Ellipse (900,186 15x15), colour toggle: m_Instance.ptrGuiCH^.stat.stState.bMOVEMENT_FAILED
    Label (760,80 140x30), "Streaming"
    Ellipse (900,86 15x15), colour toggle: m_Instance.ptrGuiCH^.stat.stState.bIS_STREAMING
    Label (760,205 140x30), "Overload"
    Ellipse (900,211 15x15), colour toggle: m_Instance.ptrGuiCH^.stat.stState.bPOSITIONER_OVERLOAD
    Label (760,230 140x30), "Overtemperature"
    Ellipse (900,236 15x15), colour toggle: m_Instance.ptrGuiCH^.stat.stState.bOVER_TEMPERATURE
    Label (560,280 140x30), "Phased"
    Ellipse (700,286 15x15), colour toggle: m_Instance.ptrGuiCH^.stat.stState.bIS_PHASED
    Label (760,255 140x30), "Positioner Fault"
    Ellipse (900,261 15x15), colour toggle: m_Instance.ptrGuiCH^.stat.stState.bPOSITIONER_FAULT
    Label (760,55 140x30), "Move Delayed"
    Ellipse (900,61 15x15), colour toggle: m_Instance.ptrGuiCH^.stat.stState.bMOVE_DELAYED
    Ellipse (120,368 20x20), tooltip "GREEN if initialised", colour toggle: m_Instance.ptrGuiCH^.stat.bInitialised
    Rectangle (145,224 325x37), "%s", tooltip "Positioner Status", text variable: m_Instance.ptrGuiCH^.stat.sStatus
    Rectangle (145,150 325x37), "%s", tooltip "Positioner Device State", text variable: m_Instance.ptrGuiCH^.stat.sState
    Rectangle (145,187 325x37), "%s", tooltip "Positioner Device Substate", text variable: m_Instance.ptrGuiCH^.stat.sSubstate
    Label (29,153 110x30), "State:"
    Label (29,190 110x30), "Substate:"
    Label (29,227 110x30), "Status:"
    Rectangle (30,17 90x30), "Ver. %s", tooltip "SmarAct Library Version", text variable: m_Instance.stat.sLibVersion
    Label (633,18 196x30), "Channel State"
    Rectangle (477,111 59x30), "%s", tooltip "Positioner User Units", text variable: m_Instance.ptrGuiCH^.cfg.sUnits
    Checkbox (470,21 116x30), "Local Control", variable: m_Instance.ptrGuiCH^.stat.bLocal
    Rectangle (145,261 325x37), "%s", tooltip "Positioner Status", text variable: m_Instance.ptrGuiCH^.stat.sRpcErrorText
    Label (29,264 110x30), "RPC Status:"
    Button (150,325 140x30), "RESET", input disabled if: NOT m_Instance.ptrGuiCH^.stat.bLocal
        OnMouseClick: execute { m_Instance.ptrGuiCH^.ctrl.nCmd:=E_SA_CH_CMD.RESET; }
    Label (567,436 130x30), "Rel Pos [UU]:"
    Rectangle (696,436 85x30), "%.3f", tooltip "Set Position Offset [UU]", text variable: m_Instance.ptrGuiCH^.ctrl.lrOff
        OnMouseClick: write the text variable via Default
    Button (329,445 140x30), "MOVE REL", input disabled if: NOT m_Instance.ptrGuiCH^.stat.bLocal OR m_Instance.ptrGuiCH^.stat.nState <> E_SA_POS_ELT_STATE.OP
        OnMouseClick: execute { m_Instance.ptrGuiCH^.ctrl.lrPos := m_Instance.ptrGuiCH^.stat.lrPosActual + m_Instance.ptrGuiCH^.ctrl.lrOff; m_Instance.ptrGuiCH^.ctrl.nCmd:=E_SA_CH_CMD.MOV; }
    Button (150,405 140x30), "ENABLE", input disabled if: NOT m_Instance.ptrGuiCH^.stat.bLocal or NOT m_Instance.ptrGuiCH^.stat.bInitialised OR m_Instance.ptrGuiCH^.stat.nState = E_SA_POS_ELT_STATE.OP
        OnMouseClick: execute { m_Instance.ptrGuiCH^.ctrl.nCmd:=E_SA_CH_CMD.ENABLE; }
    Button (329,405 140x30), "DISABLE", input disabled if: NOT m_Instance.ptrGuiCH^.stat.bLocal OR m_Instance.ptrGuiCH^.stat.nState <> E_SA_POS_ELT_STATE.OP
        OnMouseClick: execute { m_Instance.ptrGuiCH^.ctrl.nCmd:=E_SA_CH_CMD.DISABLE; }
END_VISUALIZATION
